PROGRAM PILSv2
VAR
    fbTonStartDelay: TON;
    bPILSV2isInitialized: BOOL := FALSE;
END_VAR

fbTonStartDelay(IN:=TRUE,PT:=T#4S);
IF fbTonStartDelay.Q THEN
    PILS_DEVICES();
    bPILSV2isInitialized := TRUE;
END_IF
INDEXER_COMM();

END_PROGRAM

(* stored: Version 1.1.0.1, ProductVersion 3.1.4024.11
   POU PILSv2: Id {90d527b3-98ed-47d0-a704-81d6444f3844}, SpecialFunc None *)
